// TIA Portal V17 export
// export: Created 2023-12-22T15:05:35.7408938Z, ExportSetting WithDefaults, DisplayName Totally Integrated Automation Portal, DisplayVersion V17, DisplayName TIA Portal Openness, DisplayVersion V17, DisplayName TIA Portal Version Control Interface, DisplayVersion V17, DisplayName STEP 7 Professional, DisplayVersion V17, DisplayName STEP 7 Safety, DisplayVersion V17, DisplayName WinCC Advanced, DisplayVersion V17
TYPE "PolyMix_Input"
// stored: IsFailsafeCompliant false
   STRUCT
      WatchDog : Int;
      Clock : Bool;
      Start : Bool;   // Команда запуска
      SP_C : Real;   // Уставка концентрации
      Weight : Real;
      res_1 : Real;
      res_2 : Real;
   END_STRUCT;
END_TYPE
